FUNCTION_BLOCK TcoDataManager EXTENDS TcoData.TcoDataExchange
VAR
    _data : Data;
END_VAR

END_FUNCTION_BLOCK

(* stored: Version 1.1.0.1, ProductVersion 3.1.4024.9
   POU TcoDataManager: Id {cbedc24e-3653-0ddc-2b27-80848f6cc570}, SpecialFunc None *)
